INTERFACE I_EnumDatatype EXTENDS I_UserDefinedDatatype

END_INTERFACE

(* stored: Version 1.1.0.1, ProductVersion 3.1.4024.12
   Itf I_EnumDatatype: Id {89587be6-7e6a-096a-2593-84d2b84b6449} *)
